// LS Electric XG5000 project: 동남101
// PLC NewPLC
// module base 0 slot 0: 입출력 모듈:XBC-DN/DP14E (DC 24V 입력 8점, 트랜지스터 출력 6점)

PROGRAM NewProgram (task: 스캔 프로그램)

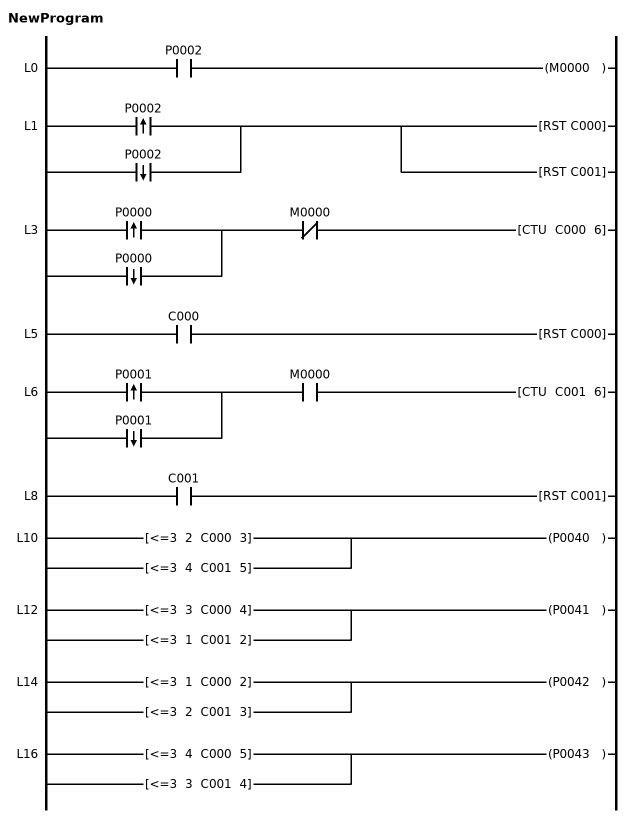
; L0
LOAD      P0002
OUT       M0000
; L1
LOADP     P0002
ORN       P0002
RST       C000
RST       C001
; L3
LOADP     P0000
ORN       P0000
AND NOT   M0000
CTU       C000 6
; L5
LOAD      C000
RST       C000
; L6
LOADP     P0001
ORN       P0001
AND       M0000
CTU       C001 6
; L8
LOAD      C001
RST       C001
; L10
LOAD<=3   2 C000 3
OR<=3     4 C001 5
OUT       P0040
; L12
LOAD<=3   3 C000 4
OR<=3     1 C001 2
OUT       P0041
; L14
LOAD<=3   1 C000 2
OR<=3     2 C001 3
OUT       P0042
; L16
LOAD<=3   4 C000 5
OR<=3     3 C001 4
OUT       P0043